// Core §7.7(c) — FB_LocalAccessProvider table entry (local default; server-side
// auth substitutes via I_AccessProvider without touching module code). Packed:
// it is also the record of the retained ST_AccessImageV1.
{attribute 'pack_mode' := '1'}
TYPE ST_UserRecord :
STRUCT
    User    : STRING(32);
    // §14 - the PIN itself is never stored: a salt drawn at registration and the
    // iterated SHA-256 of salt and PIN (FB_LocalAccessProvider._M_Hash).
    Salt    : ARRAY[0..15] OF BYTE;
    PinHash : ARRAY[0..31] OF BYTE;
    Level   : E_AccessLevel;
END_STRUCT
END_TYPE

(* stored: Version 1.1.0.1, ProductVersion 3.1.4024.12
   DUT ST_UserRecord: Id {224b60fd-3441-4d16-98a8-4792000f9df1} *)
